PROGRAM MRU2
VAR
	buffer			: ARRAY [1..1024] OF BYTE;
	_feedback		: MruFeedback;
	
	NULL			: PVOID;
	UdpIO			: UdpServer(7552, 0, NULL, SIZEOF(_feedback), ADR(buffer));
		
	temp			: ARRAY [0..3] OF BYTE;
	N				: DINT;
END_VAR

VAR_OUTPUT
	feedback		: RemoteFeedbackMru;
END_VAR


UdpIO();

_feedback.mruOK := buffer[1];
_feedback.dataLength := buffer[2];
_feedback.token := buffer[3];


// Big to little endian conversions
N := 1;
temp[3] := buffer[N*4];
temp[2] := buffer[N*4 + 1];
temp[1] := buffer[N*4 + 2];
temp[0] := buffer[N*4 + 3]; 
MEMCPY(ADR(_feedback.Temperature), ADR(temp), 4);

N := 2;
temp[3] := buffer[N*4];
temp[2] := buffer[N*4 + 1];
temp[1] := buffer[N*4 + 2];
temp[0] := buffer[N*4 + 3]; 
MEMCPY(ADR(_feedback.PosMru_D), ADR(temp), 4);

N := 3;
temp[3] := buffer[N*4];
temp[2] := buffer[N*4 + 1];
temp[1] := buffer[N*4 + 2];
temp[0] := buffer[N*4 + 3];
MEMCPY(ADR(_feedback.VelMru_D), ADR(temp), 4);

N := 4;
temp[3] := buffer[N*4];
temp[2] := buffer[N*4 + 1];
temp[1] := buffer[N*4 + 2];
temp[0] := buffer[N*4 + 3];
MEMCPY(ADR(_feedback.AccMru_D), ADR(temp), 4);

N := 5;
temp[3] := buffer[N*4];
temp[2] := buffer[N*4 + 1];
temp[1] := buffer[N*4 + 2];
temp[0] := buffer[N*4 + 3];
MEMCPY(ADR(_feedback.AngRate_D), ADR(temp), 4);

N := 6;
temp[3] := buffer[N*4];
temp[2] := buffer[N*4 + 1];
temp[1] := buffer[N*4 + 2];
temp[0] := buffer[N*4 + 3];
MEMCPY(ADR(_feedback.Roll), ADR(temp), 4);

N := 7;
temp[3] := buffer[N*4];
temp[2] := buffer[N*4 + 1];
temp[1] := buffer[N*4 + 2];
temp[0] := buffer[N*4 + 3];
MEMCPY(ADR(_feedback.Pitch), ADR(temp), 4);

N := 8;
temp[3] := buffer[N*4];
temp[2] := buffer[N*4 + 1];
temp[1] := buffer[N*4 + 2];
temp[0] := buffer[N*4 + 3];
MEMCPY(ADR(_feedback.Yaw), ADR(temp), 4);

N := 9;
temp[3] := buffer[N*4];
temp[2] := buffer[N*4 + 1];
temp[1] := buffer[N*4 + 2];
temp[0] := buffer[N*4 + 3];
MEMCPY(ADR(_feedback.AngRate_R), ADR(temp), 4);

N := 10;
temp[3] := buffer[N*4];
temp[2] := buffer[N*4 + 1];
temp[1] := buffer[N*4 + 2];
temp[0] := buffer[N*4 + 3];
MEMCPY(ADR(_feedback.AngRate_P), ADR(temp), 4);

N := 11;
temp[3] := buffer[N*4];
temp[2] := buffer[N*4 + 1];
temp[1] := buffer[N*4 + 2];
temp[0] := buffer[N*4 + 3];
MEMCPY(ADR(_feedback.AngRate_Y), ADR(temp), 4);

N := 12;
temp[3] := buffer[N*4];
temp[2] := buffer[N*4 + 1];
temp[1] := buffer[N*4 + 2];
temp[0] := buffer[N*4 + 3];
MEMCPY(ADR(_feedback.AngAcc_R), ADR(temp), 4);

N := 13;
temp[3] := buffer[N*4];
temp[2] := buffer[N*4 + 1];
temp[1] := buffer[N*4 + 2];
temp[0] := buffer[N*4 + 3];
MEMCPY(ADR(_feedback.AngAcc_P), ADR(temp), 4);

N := 14;
temp[3] := buffer[N*4];
temp[2] := buffer[N*4 + 1];
temp[1] := buffer[N*4 + 2];
temp[0] := buffer[N*4 + 3];
MEMCPY(ADR(_feedback.AngAcc_Y), ADR(temp), 4);

N := 15;
temp[3] := buffer[N*4];
temp[2] := buffer[N*4 + 1];
temp[1] := buffer[N*4 + 2];
temp[0] := buffer[N*4 + 3];
MEMCPY(ADR(_feedback.VelMru_R), ADR(temp), 4);

N := 16;
temp[3] := buffer[N*4];
temp[2] := buffer[N*4 + 1];
temp[1] := buffer[N*4 + 2];
temp[0] := buffer[N*4 + 3];
MEMCPY(ADR(_feedback.VelMru_P), ADR(temp), 4);

N := 17;
temp[3] := buffer[N*4];
temp[2] := buffer[N*4 + 1];
temp[1] := buffer[N*4 + 2];
temp[0] := buffer[N*4 + 3];
MEMCPY(ADR(_feedback.VelMru_Y), ADR(temp), 4);

N := 18;
temp[3] := buffer[N*4];
temp[2] := buffer[N*4 + 1];
temp[1] := buffer[N*4 + 2];
temp[0] := buffer[N*4 + 3];
MEMCPY(ADR(_feedback.AccMru_R), ADR(temp), 4);

N := 19;
temp[3] := buffer[N*4];
temp[2] := buffer[N*4 + 1];
temp[1] := buffer[N*4 + 2];
temp[0] := buffer[N*4 + 3];
MEMCPY(ADR(_feedback.AccMru_P), ADR(temp), 4);

N := 20;
temp[3] := buffer[N*4];
temp[2] := buffer[N*4 + 1];
temp[1] := buffer[N*4 + 2];
temp[0] := buffer[N*4 + 3];
MEMCPY(ADR(_feedback.AccMru_Y), ADR(temp), 4);

// Convert data to remote feedback
feedback.heave := _feedback.PosMru_D;
feedback.heave_t := _feedback.VelMru_D;
feedback.heave_tt := _feedback.AccMru_D;
feedback.turn_rate := _feedback.AngRate_D;
feedback.roll := _feedback.Roll;
feedback.pitch := _feedback.Pitch;
feedback.yaw := _feedback.Yaw;
feedback.wx := _feedback.AngRate_R;
feedback.wy := _feedback.AngRate_P;
feedback.wz := _feedback.AngRate_Y;
feedback.wx_t := _feedback.AngAcc_R;
feedback.wy_t := _feedback.AngAcc_P;
feedback.wz_t := _feedback.AngAcc_Y;
feedback.x_t := _feedback.VelMru_R;
feedback.y_t := _feedback.VelMru_P;
feedback.z_t := _feedback.VelMru_Y;
feedback.x_tt := _feedback.AccMru_R;
feedback.y_tt := _feedback.AccMru_P;
feedback.z_tt := _feedback.AccMru_Y;

END_PROGRAM

(* stored: Version 1.1.0.1, ProductVersion 3.1.4020.12
   POU MRU2: Id {76aeb5d9-7025-4781-8e97-1cc2a072ff52}, SpecialFunc None *)
